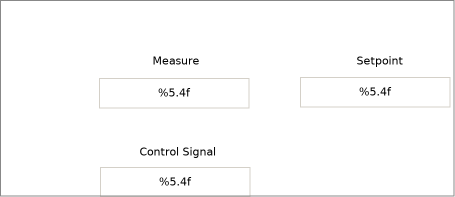
VISUALIZATION VISU1  // 455x197
    Textfield (99,78 150x30), "%5.4f", text variable: MAIN.AIN1
    Textfield (100,167 150x30), "%5.4f", text variable: MAIN.OUT
    Label (101,46 150x30), "Measure"
    Label (103,137 150x30), "Control Signal"
    Textfield (300,77 150x30), "%5.4f", text variable: PID_DATA.gset
    Label (305,46 150x30), "Setpoint"
END_VISUALIZATION

(* stored: Version 1.1.0.1, ProductVersion 3.1.4024.3
   Visu VISU1: Id {a7643927-47da-4809-a06e-e1553d38f97d} *)
